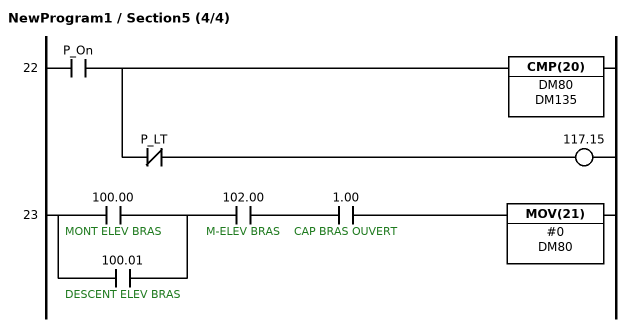
; [picture p24: NewProgram1 / Section5, rungs 22-23]
; rung 22
LD P_On
CMP(20) DM80 DM135
ANDNOT P_LT
OUT 117.15
; rung 23
LD 100.00  ; MONT ELEV BRAS
OR 100.01  ; DESCENT ELEV BRAS
AND 102.00  ; M-ELEV BRAS
AND 1.00  ; CAP BRAS OUVERT
MOV(21) #0 DM80

### Section Section6

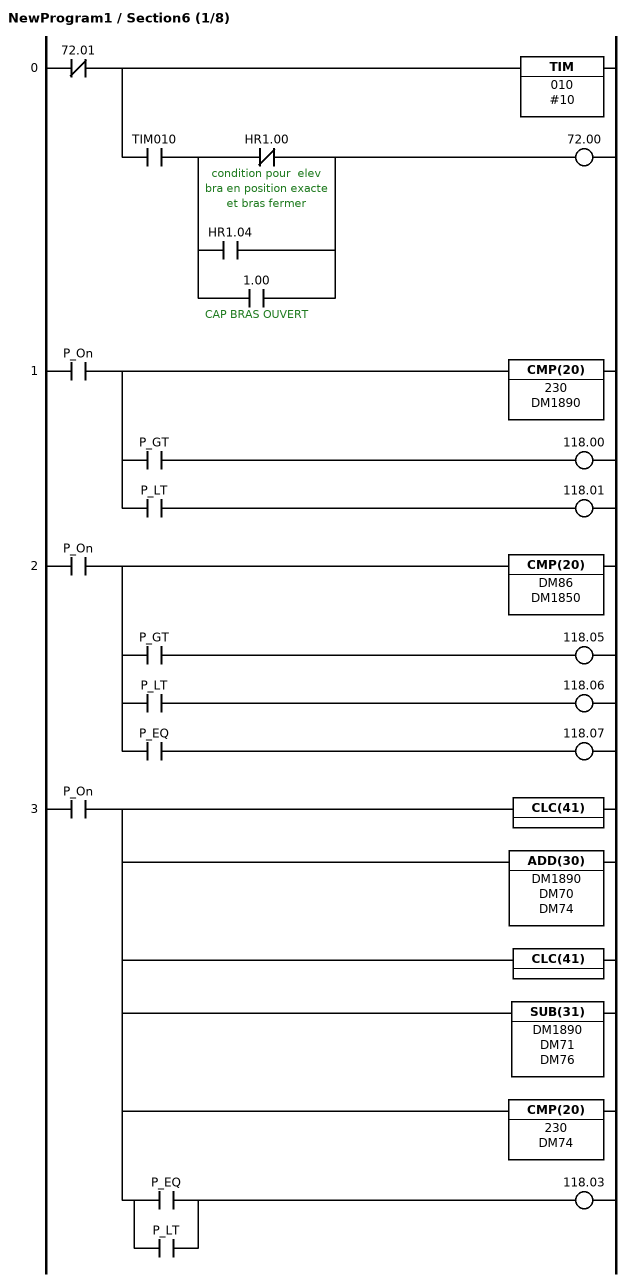
; rung 0
LDNOT 72.01
TIM 010 #10
AND TIM010
LDNOT HR1.00  ; condition pour  elev bra en position exacte et bras fermer
OR HR1.04
OR 1.00  ; CAP BRAS OUVERT
ANDLD
OUT 72.00
; rung 1
LD P_On
OUT TR0
CMP(20) 230 DM1890
AND P_GT
OUT 118.00
LD TR0
AND P_LT
OUT 118.01
; rung 2
LD P_On
OUT TR0
CMP(20) DM86 DM1850
AND P_GT
OUT 118.05
LD TR0
AND P_LT
OUT 118.06
LD TR0
AND P_EQ
OUT 118.07
; rung 3
LD P_On
CLC(41)
ADD(30) DM1890 DM70 DM74
CLC(41)
SUB(31) DM1890 DM71 DM76
CMP(20) 230 DM74
LD P_EQ
OR P_LT
ANDLD
OUT 118.03

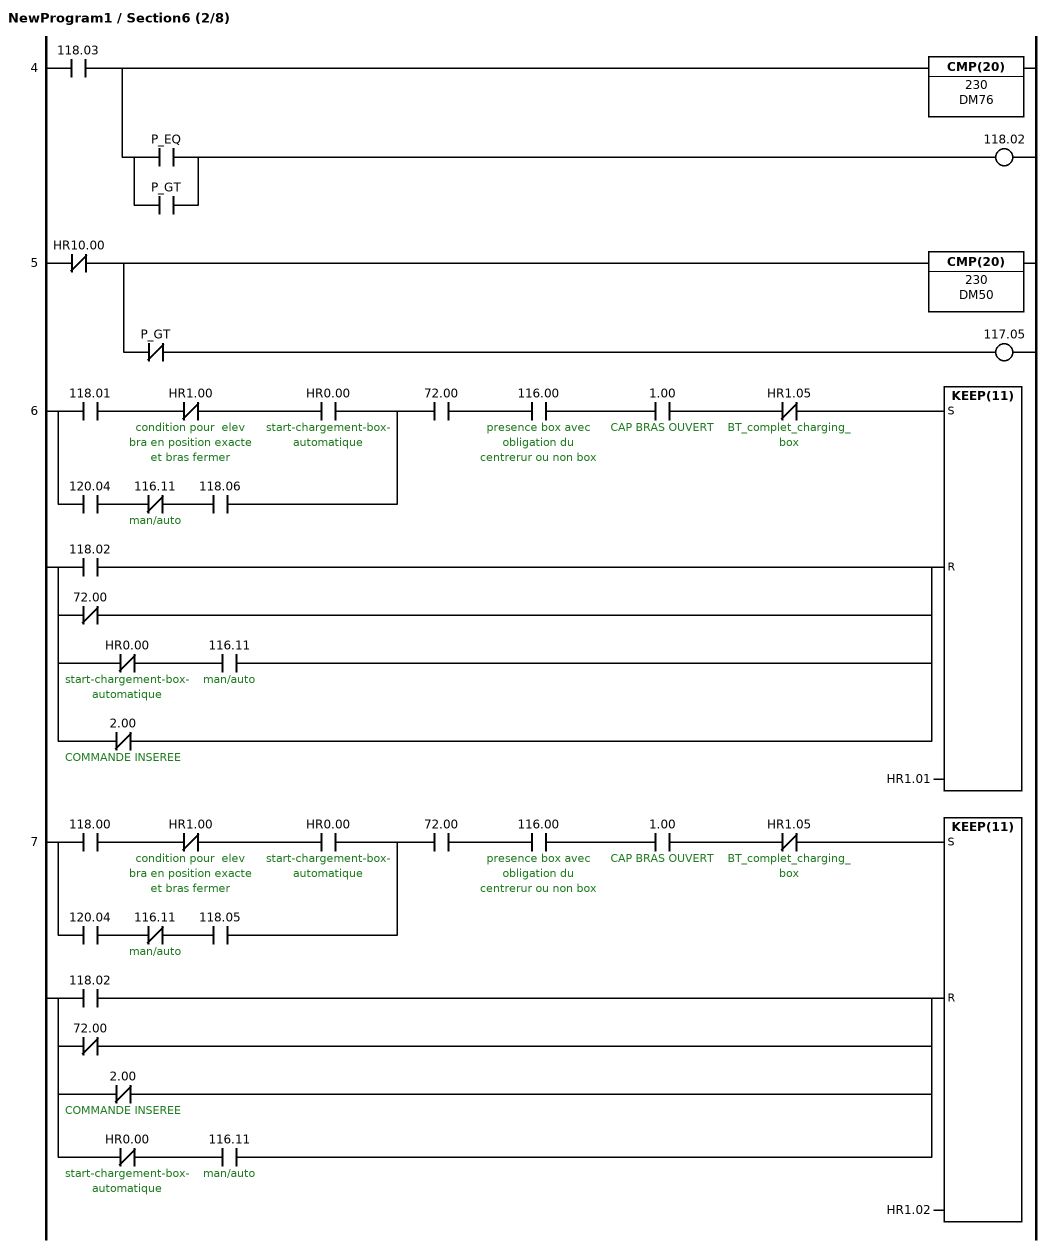
; rung 4
LD 118.03
CMP(20) 230 DM76
LD P_EQ
OR P_GT
ANDLD
OUT 118.02
; rung 5
LDNOT HR10.00
CMP(20) 230 DM50
ANDNOT P_GT
OUT 117.05
; rung 6
LD 118.01
ANDNOT HR1.00  ; condition pour  elev bra en position exacte et bras fermer
AND HR0.00  ; start-chargement-box-automatique
LD 120.04
ANDNOT 116.11  ; man/auto
AND 118.06
ORLD
AND 72.00
AND 116.00  ; presence box avec obligation du centrerur ou non box
AND 1.00  ; CAP BRAS OUVERT
ANDNOT HR1.05  ; BT_complet_charging_box
LD 118.02
ORNOT 72.00
LDNOT HR0.00  ; start-chargement-box-automatique
AND 116.11  ; man/auto
ORLD
ORNOT 2.00  ; COMMANDE INSEREE
KEEP(11) HR1.01
; rung 7
LD 118.00
ANDNOT HR1.00  ; condition pour  elev bra en position exacte et bras fermer
AND HR0.00  ; start-chargement-box-automatique
LD 120.04
ANDNOT 116.11  ; man/auto
AND 118.05
ORLD
AND 72.00
AND 116.00  ; presence box avec obligation du centrerur ou non box
AND 1.00  ; CAP BRAS OUVERT
ANDNOT HR1.05  ; BT_complet_charging_box
LD 118.02
ORNOT 72.00
ORNOT 2.00  ; COMMANDE INSEREE
LDNOT HR0.00  ; start-chargement-box-automatique
AND 116.11  ; man/auto
ORLD
KEEP(11) HR1.02

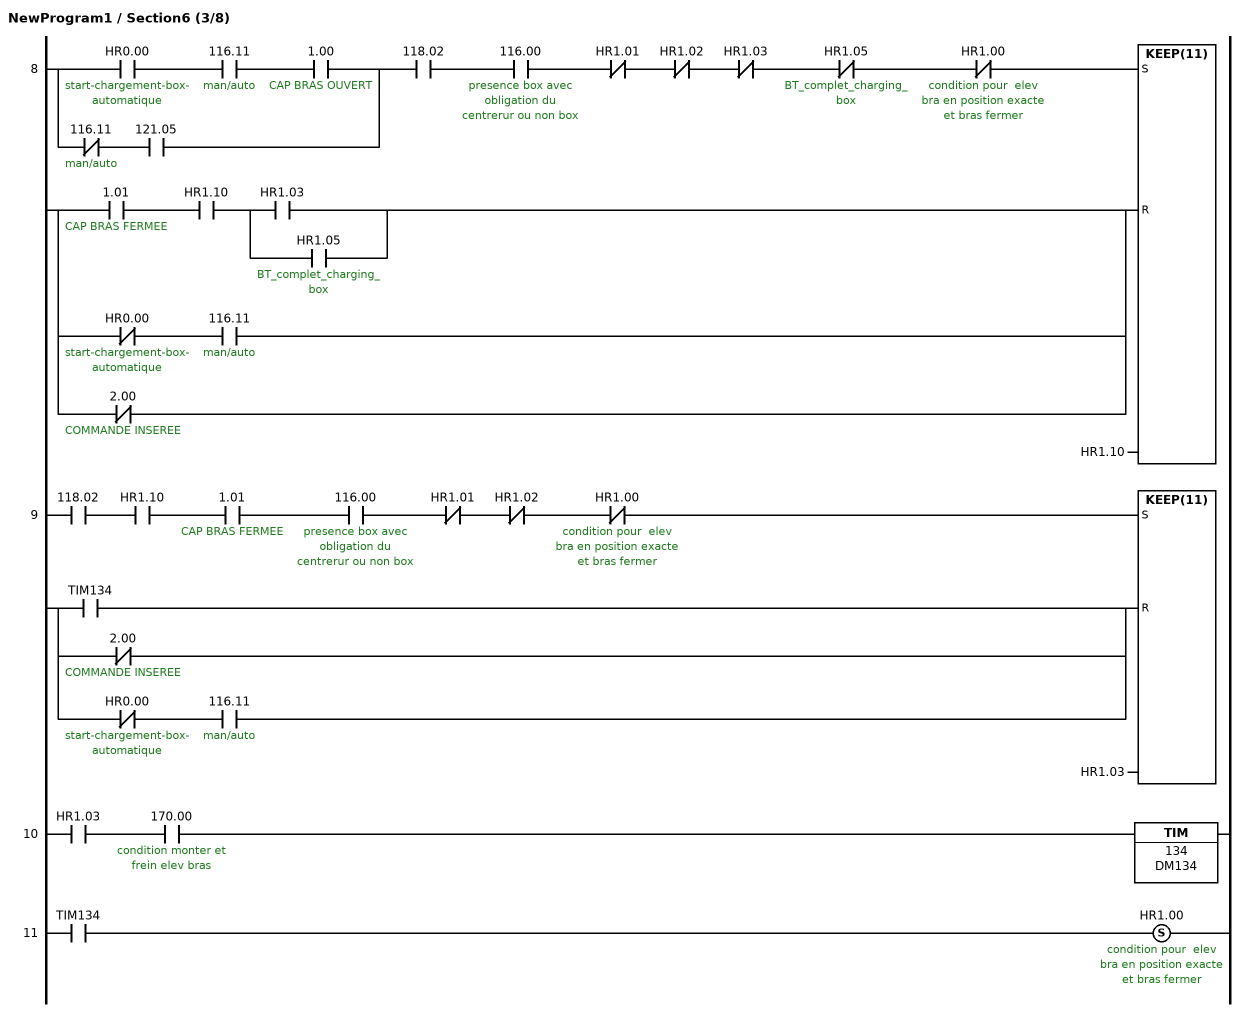
; rung 8
LD HR0.00  ; start-chargement-box-automatique
AND 116.11  ; man/auto
AND 1.00  ; CAP BRAS OUVERT
LDNOT 116.11  ; man/auto
AND 121.05
ORLD
AND 118.02
AND 116.00  ; presence box avec obligation du centrerur ou non box
ANDNOT HR1.01
ANDNOT HR1.02
ANDNOT HR1.03
ANDNOT HR1.05  ; BT_complet_charging_box
ANDNOT HR1.00  ; condition pour  elev bra en position exacte et bras fermer
LD 1.01  ; CAP BRAS FERMEE
AND HR1.10
LD HR1.03
OR HR1.05  ; BT_complet_charging_box
ANDLD
LDNOT HR0.00  ; start-chargement-box-automatique
AND 116.11  ; man/auto
ORLD
ORNOT 2.00  ; COMMANDE INSEREE
KEEP(11) HR1.10
; rung 9
LD 118.02
AND HR1.10
AND 1.01  ; CAP BRAS FERMEE
AND 116.00  ; presence box avec obligation du centrerur ou non box
ANDNOT HR1.01
ANDNOT HR1.02
ANDNOT HR1.00  ; condition pour  elev bra en position exacte et bras fermer
LD TIM134
ORNOT 2.00  ; COMMANDE INSEREE
LDNOT HR0.00  ; start-chargement-box-automatique
AND 116.11  ; man/auto
ORLD
KEEP(11) HR1.03
; rung 10
LD HR1.03
AND 170.00  ; condition monter et frein elev bras
TIM 134 DM134
; rung 11
LD TIM134
SET HR1.00  ; condition pour  elev bra en position exacte et bras fermer

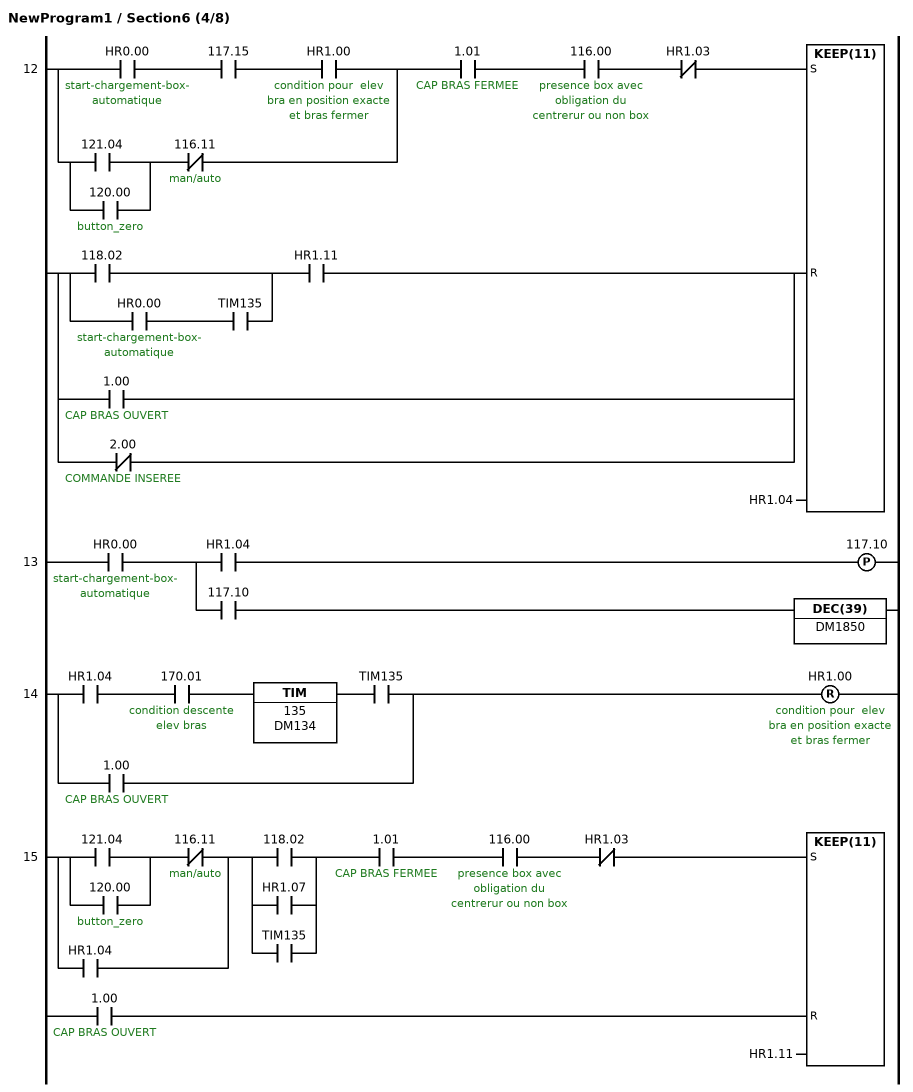
; rung 12
LD HR0.00  ; start-chargement-box-automatique
AND 117.15
AND HR1.00  ; condition pour  elev bra en position exacte et bras fermer
LD 121.04
OR 120.00  ; button_zero
ANDNOT 116.11  ; man/auto
ORLD
AND 1.01  ; CAP BRAS FERMEE
AND 116.00  ; presence box avec obligation du centrerur ou non box
ANDNOT HR1.03
LD 118.02
LD HR0.00  ; start-chargement-box-automatique
AND TIM135
ORLD
AND HR1.11
OR 1.00  ; CAP BRAS OUVERT
ORNOT 2.00  ; COMMANDE INSEREE
KEEP(11) HR1.04
; rung 13
LD HR0.00  ; start-chargement-box-automatique
OUT TR0
AND HR1.04
DIFU(13) 117.10
LD TR0
AND 117.10
DEC(39) DM1850
; rung 14
LD HR1.04
AND 170.01  ; condition descente elev bras
TIM 135 DM134
AND TIM135
OR 1.00  ; CAP BRAS OUVERT
RSET HR1.00  ; condition pour  elev bra en position exacte et bras fermer
; rung 15
LD 121.04
OR 120.00  ; button_zero
ANDNOT 116.11  ; man/auto
OR HR1.04
LD 118.02
OR HR1.07
OR TIM135
ANDLD
AND 1.01  ; CAP BRAS FERMEE
AND 116.00  ; presence box avec obligation du centrerur ou non box
ANDNOT HR1.03
LD 1.00  ; CAP BRAS OUVERT
KEEP(11) HR1.11

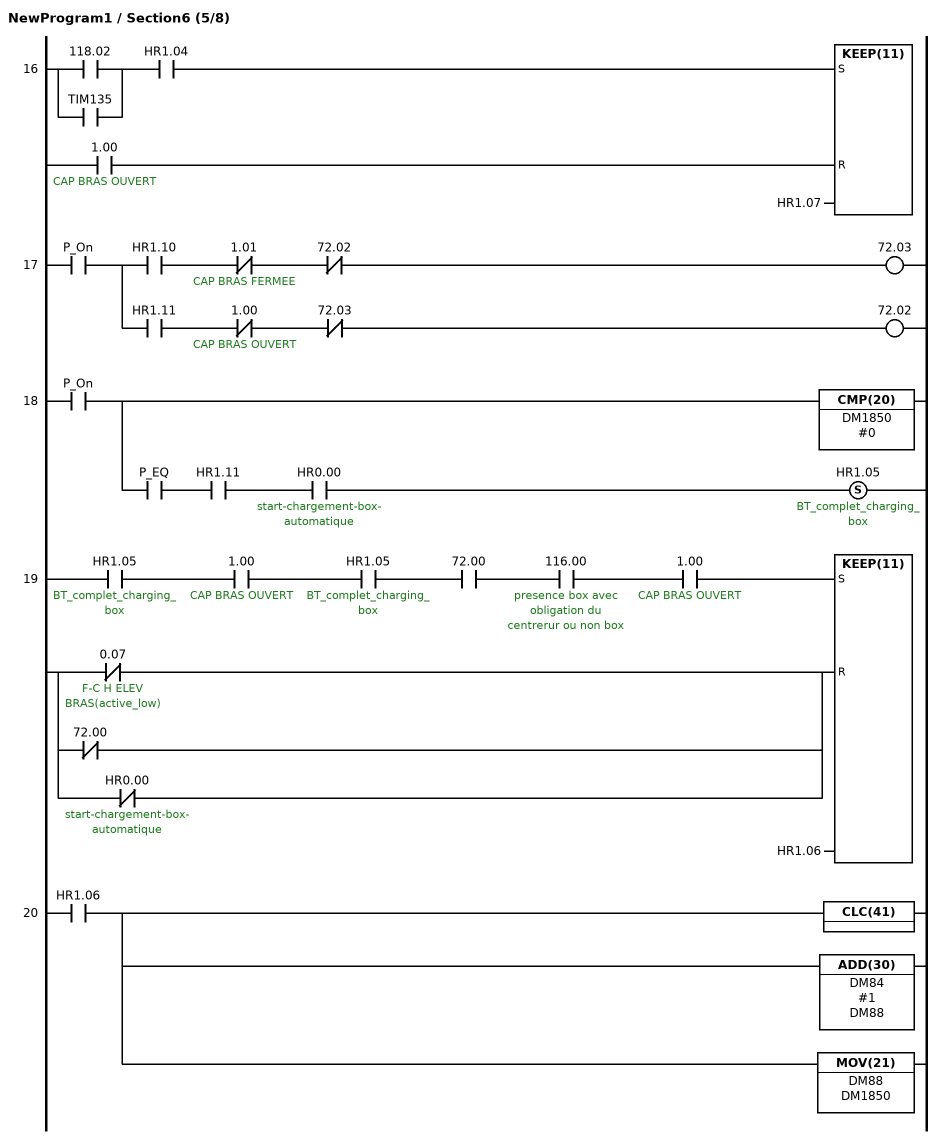
; rung 16
LD 118.02
OR TIM135
AND HR1.04
LD 1.00  ; CAP BRAS OUVERT
KEEP(11) HR1.07
; rung 17
LD P_On
OUT TR0
AND HR1.10
ANDNOT 1.01  ; CAP BRAS FERMEE
ANDNOT 72.02
OUT 72.03
LD TR0
AND HR1.11
ANDNOT 1.00  ; CAP BRAS OUVERT
ANDNOT 72.03
OUT 72.02
; rung 18
LD P_On
CMP(20) DM1850 #0
AND P_EQ
AND HR1.11
AND HR0.00  ; start-chargement-box-automatique
SET HR1.05  ; BT_complet_charging_box
; rung 19
LD HR1.05  ; BT_complet_charging_box
AND 1.00  ; CAP BRAS OUVERT
AND HR1.05  ; BT_complet_charging_box
AND 72.00
AND 116.00  ; presence box avec obligation du centrerur ou non box
AND 1.00  ; CAP BRAS OUVERT
LDNOT 0.07  ; F-C H ELEV BRAS(active_low)
ORNOT 72.00
ORNOT HR0.00  ; start-chargement-box-automatique
KEEP(11) HR1.06
; rung 20
LD HR1.06
CLC(41)
ADD(30) DM84 #1 DM88
MOV(21) DM88 DM1850

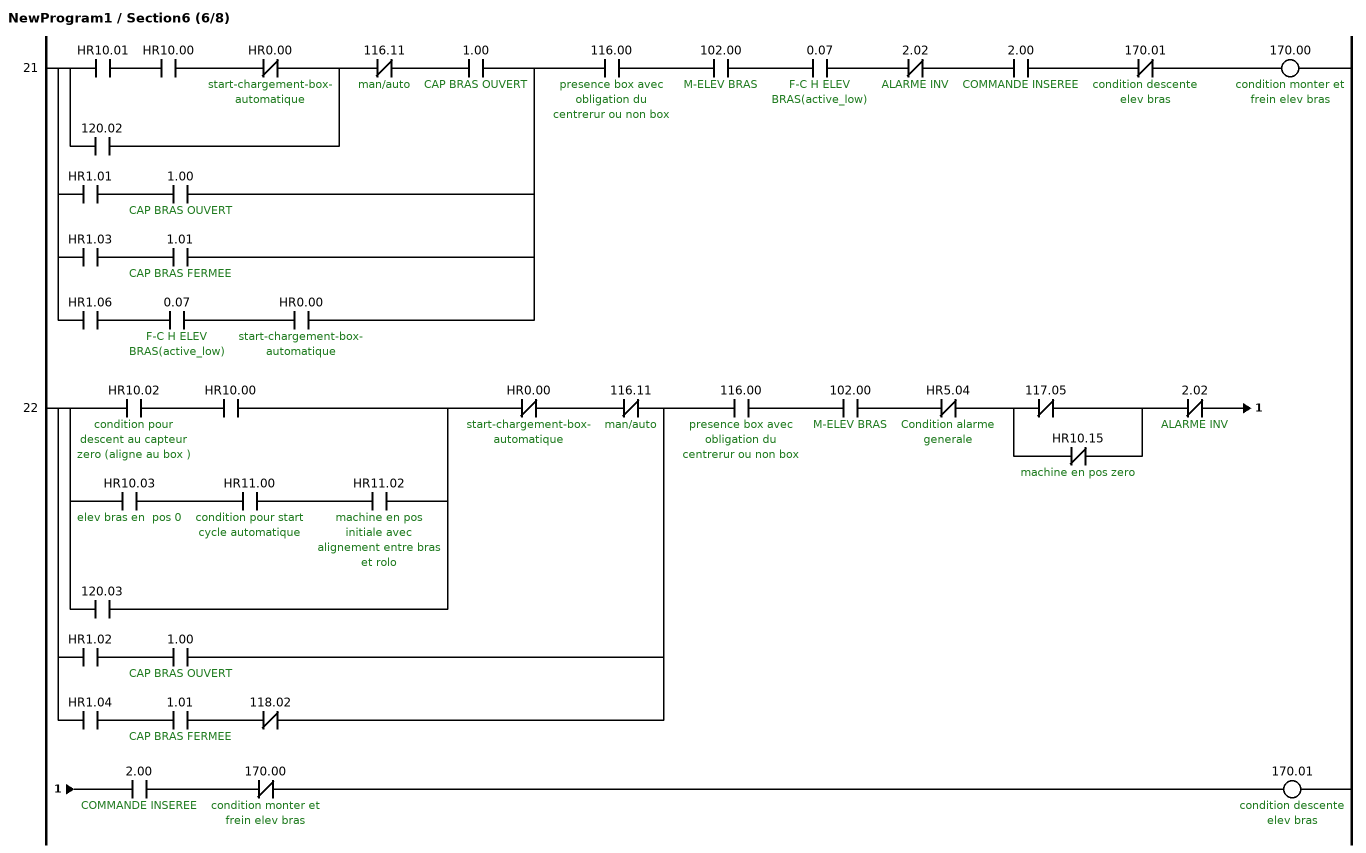
; rung 21
LD HR10.01
AND HR10.00
ANDNOT HR0.00  ; start-chargement-box-automatique
OR 120.02
ANDNOT 116.11  ; man/auto
AND 1.00  ; CAP BRAS OUVERT
LD HR1.01
AND 1.00  ; CAP BRAS OUVERT
ORLD
LD HR1.03
AND 1.01  ; CAP BRAS FERMEE
ORLD
LD HR1.06
AND 0.07  ; F-C H ELEV BRAS(active_low)
AND HR0.00  ; start-chargement-box-automatique
ORLD
AND 116.00  ; presence box avec obligation du centrerur ou non box
AND 102.00  ; M-ELEV BRAS
AND 0.07  ; F-C H ELEV BRAS(active_low)
ANDNOT 2.02  ; ALARME INV
AND 2.00  ; COMMANDE INSEREE
ANDNOT 170.01  ; condition descente elev bras
OUT 170.00  ; condition monter et frein elev bras
; rung 22
LD HR10.02  ; condition pour descent au capteur zero (aligne au box )
AND HR10.00
LD HR10.03  ; elev bras en  pos 0
AND HR11.00  ; condition pour start cycle automatique
AND HR11.02  ; machine en pos initiale avec alignement entre bras et rolo
ORLD
OR 120.03
ANDNOT HR0.00  ; start-chargement-box-automatique
ANDNOT 116.11  ; man/auto
LD HR1.02
AND 1.00  ; CAP BRAS OUVERT
ORLD
LD HR1.04
AND 1.01  ; CAP BRAS FERMEE
ANDNOT 118.02
ORLD
AND 116.00  ; presence box avec obligation du centrerur ou non box
AND 102.00  ; M-ELEV BRAS
ANDNOT HR5.04  ; Condition alarme generale
LDNOT 117.05
ORNOT HR10.15  ; machine en pos zero
ANDLD
ANDNOT 2.02  ; ALARME INV
AND 2.00  ; COMMANDE INSEREE
ANDNOT 170.00  ; condition monter et frein elev bras
OUT 170.01  ; condition descente elev bras

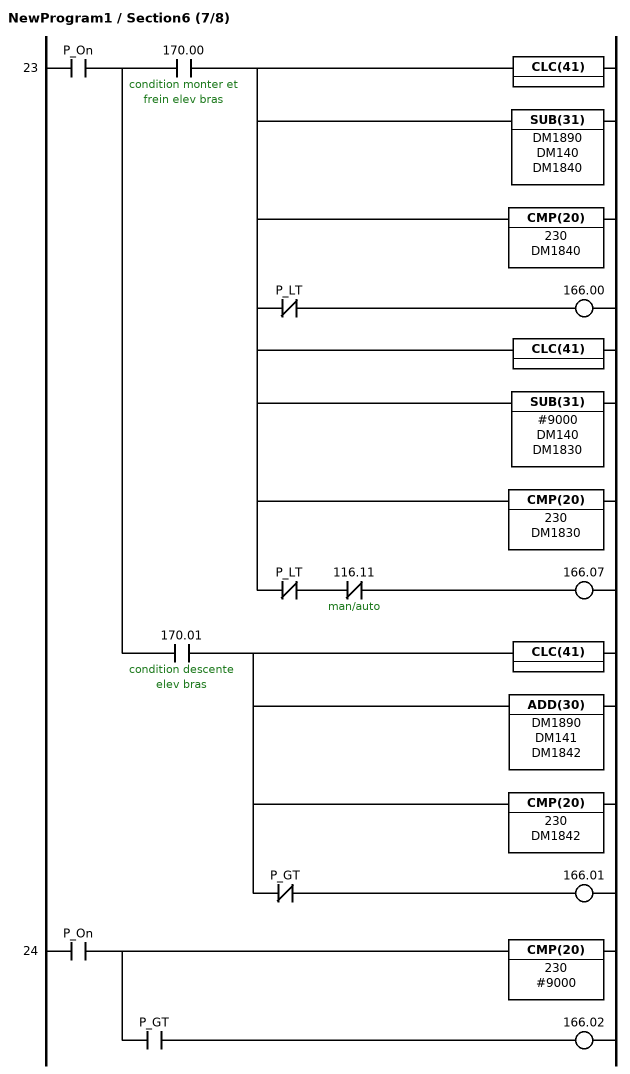
; rung 23
LD P_On
OUT TR0
AND 170.00  ; condition monter et frein elev bras
OUT TR1
CLC(41)
SUB(31) DM1890 DM140 DM1840
CMP(20) 230 DM1840
ANDNOT P_LT
OUT 166.00
LD TR1
CLC(41)
SUB(31) #9000 DM140 DM1830
CMP(20) 230 DM1830
ANDNOT P_LT
ANDNOT 116.11  ; man/auto
OUT 166.07
LD TR0
AND 170.01  ; condition descente elev bras
CLC(41)
ADD(30) DM1890 DM141 DM1842
CMP(20) 230 DM1842
ANDNOT P_GT
OUT 166.01
; rung 24
LD P_On
CMP(20) 230 #9000
AND P_GT
OUT 166.02

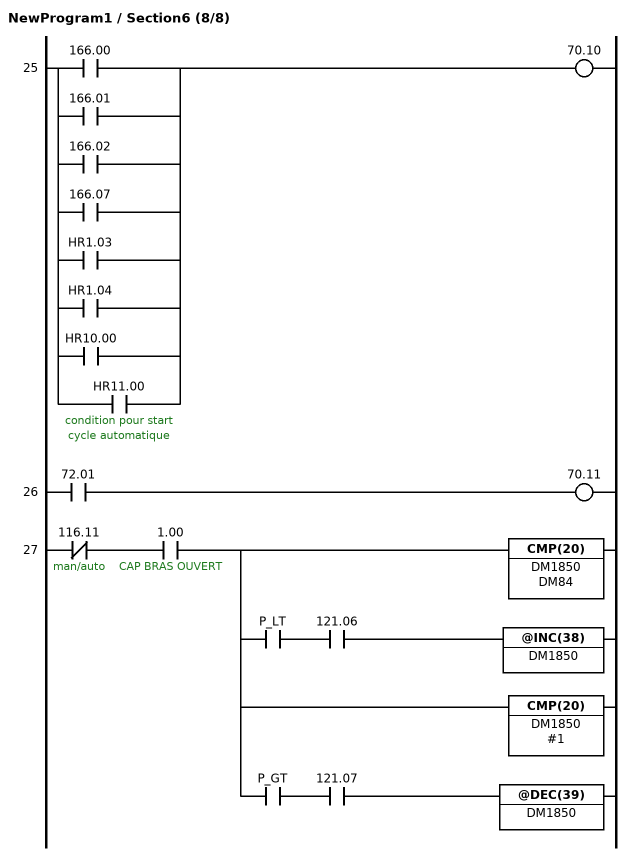
; rung 25
LD 166.00
OR 166.01
OR 166.02
OR 166.07
OR HR1.03
OR HR1.04
OR HR10.00
OR HR11.00  ; condition pour start cycle automatique
OUT 70.10
; rung 26
LD 72.01
OUT 70.11
; rung 27
LDNOT 116.11  ; man/auto
AND 1.00  ; CAP BRAS OUVERT
OUT TR0
CMP(20) DM1850 DM84
AND P_LT
AND 121.06
@INC(38) DM1850
LD TR0
CMP(20) DM1850 #1
AND P_GT
AND 121.07
@DEC(39) DM1850

### Section Section7

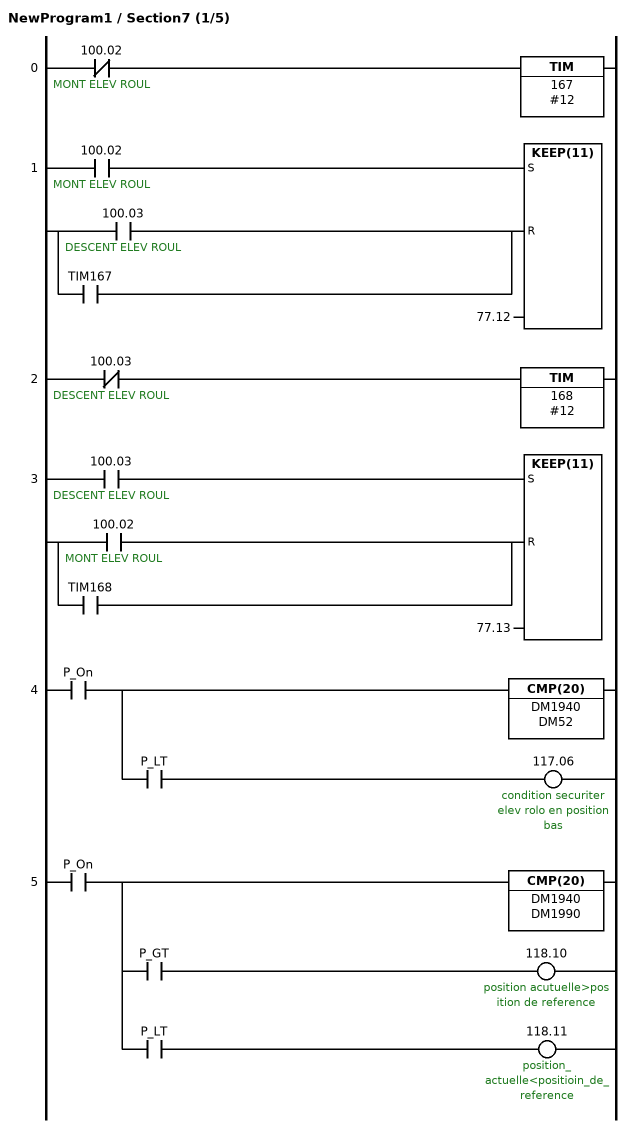
; rung 0
LDNOT 100.02  ; MONT ELEV ROUL
TIM 167 #12
; rung 1
LD 100.02  ; MONT ELEV ROUL
LD 100.03  ; DESCENT ELEV ROUL
OR TIM167
KEEP(11) 77.12
; rung 2
LDNOT 100.03  ; DESCENT ELEV ROUL
TIM 168 #12
; rung 3
LD 100.03  ; DESCENT ELEV ROUL
LD 100.02  ; MONT ELEV ROUL
OR TIM168
KEEP(11) 77.13
; rung 4
LD P_On
CMP(20) DM1940 DM52
AND P_LT
OUT 117.06  ; condition securiter elev rolo en position bas
; rung 5
LD P_On
OUT TR0
CMP(20) DM1940 DM1990
AND P_GT
OUT 118.10  ; position acutuelle>position de reference
LD TR0
AND P_LT
OUT 118.11  ; position_actuelle<positioin_de_reference

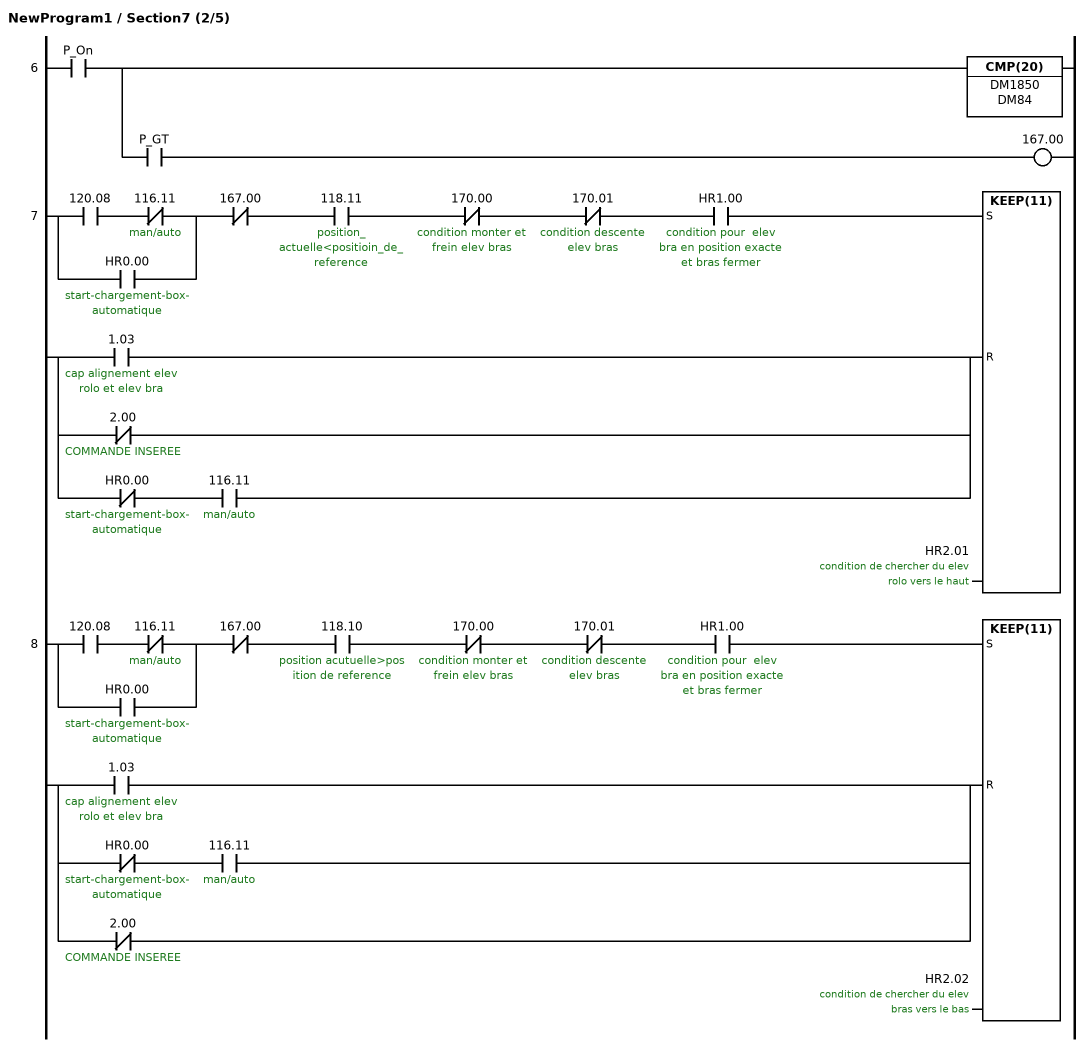
; rung 6
LD P_On
CMP(20) DM1850 DM84
AND P_GT
OUT 167.00
; rung 7
LD 120.08
ANDNOT 116.11  ; man/auto
OR HR0.00  ; start-chargement-box-automatique
ANDNOT 167.00
AND 118.11  ; position_actuelle<positioin_de_reference
ANDNOT 170.00  ; condition monter et frein elev bras
ANDNOT 170.01  ; condition descente elev bras
AND HR1.00  ; condition pour  elev bra en position exacte et bras fermer
LD 1.03  ; cap alignement elev rolo et elev bra
ORNOT 2.00  ; COMMANDE INSEREE
LDNOT HR0.00  ; start-chargement-box-automatique
AND 116.11  ; man/auto
ORLD
KEEP(11) HR2.01  ; condition de chercher du elev rolo vers le haut
; rung 8
LD 120.08
ANDNOT 116.11  ; man/auto
OR HR0.00  ; start-chargement-box-automatique
ANDNOT 167.00
AND 118.10  ; position acutuelle>position de reference
ANDNOT 170.00  ; condition monter et frein elev bras
ANDNOT 170.01  ; condition descente elev bras
AND HR1.00  ; condition pour  elev bra en position exacte et bras fermer
LD 1.03  ; cap alignement elev rolo et elev bra
LDNOT HR0.00  ; start-chargement-box-automatique
AND 116.11  ; man/auto
ORLD
ORNOT 2.00  ; COMMANDE INSEREE
KEEP(11) HR2.02  ; condition de chercher du elev bras vers le bas

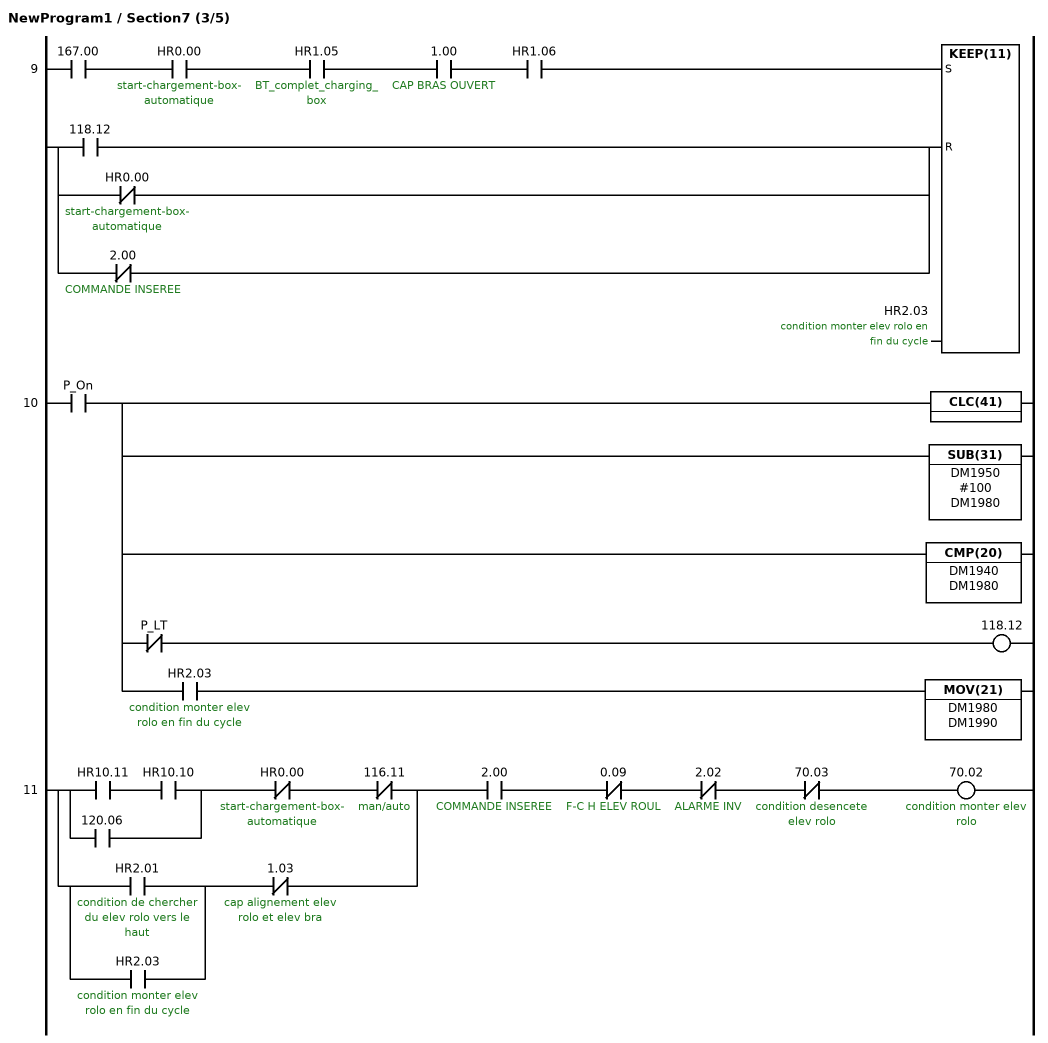
; rung 9
LD 167.00
AND HR0.00  ; start-chargement-box-automatique
AND HR1.05  ; BT_complet_charging_box
AND 1.00  ; CAP BRAS OUVERT
AND HR1.06
LD 118.12
ORNOT HR0.00  ; start-chargement-box-automatique
ORNOT 2.00  ; COMMANDE INSEREE
KEEP(11) HR2.03  ; condition monter elev rolo en fin du cycle
; rung 10
LD P_On
OUT TR0
CLC(41)
SUB(31) DM1950 #100 DM1980
CMP(20) DM1940 DM1980
ANDNOT P_LT
OUT 118.12
LD TR0
AND HR2.03  ; condition monter elev rolo en fin du cycle
MOV(21) DM1980 DM1990
; rung 11
LD HR10.11
AND HR10.10
OR 120.06
ANDNOT HR0.00  ; start-chargement-box-automatique
ANDNOT 116.11  ; man/auto
LD HR2.01  ; condition de chercher du elev rolo vers le haut
OR HR2.03  ; condition monter elev rolo en fin du cycle
ANDNOT 1.03  ; cap alignement elev rolo et elev bra
ORLD
AND 2.00  ; COMMANDE INSEREE
ANDNOT 0.09  ; F-C H ELEV ROUL
ANDNOT 2.02  ; ALARME INV
ANDNOT 70.03  ; condition desencete elev rolo
OUT 70.02  ; condition monter elev rolo

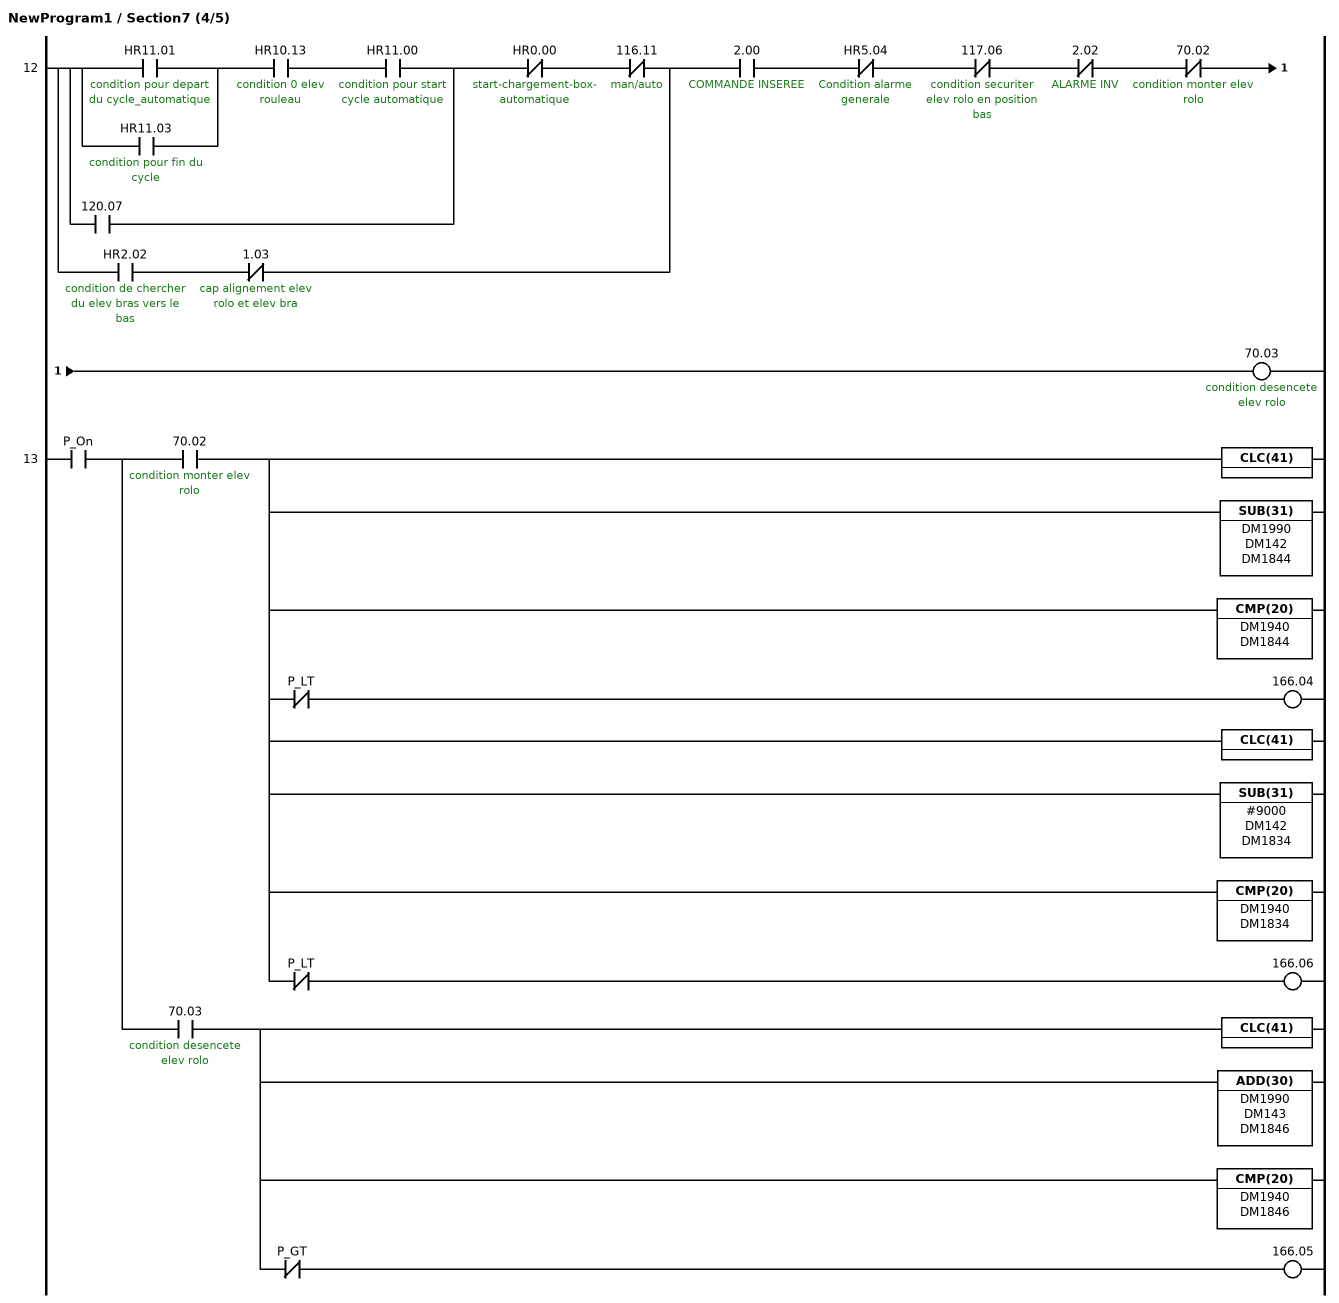
; rung 12
LD HR11.01  ; condition pour depart du cycle_automatique
OR HR11.03  ; condition pour fin du cycle
AND HR10.13  ; condition 0 elev rouleau
AND HR11.00  ; condition pour start cycle automatique
OR 120.07
ANDNOT HR0.00  ; start-chargement-box-automatique
ANDNOT 116.11  ; man/auto
LD HR2.02  ; condition de chercher du elev bras vers le bas
ANDNOT 1.03  ; cap alignement elev rolo et elev bra
ORLD
AND 2.00  ; COMMANDE INSEREE
ANDNOT HR5.04  ; Condition alarme generale
ANDNOT 117.06  ; condition securiter elev rolo en position bas
ANDNOT 2.02  ; ALARME INV
ANDNOT 70.02  ; condition monter elev rolo
OUT 70.03  ; condition desencete elev rolo
; rung 13
LD P_On
OUT TR0
AND 70.02  ; condition monter elev rolo
OUT TR1
CLC(41)
SUB(31) DM1990 DM142 DM1844
CMP(20) DM1940 DM1844
ANDNOT P_LT
OUT 166.04
LD TR1
CLC(41)
SUB(31) #9000 DM142 DM1834
CMP(20) DM1940 DM1834
ANDNOT P_LT
OUT 166.06
LD TR0
AND 70.03  ; condition desencete elev rolo
CLC(41)
ADD(30) DM1990 DM143 DM1846
CMP(20) DM1940 DM1846
ANDNOT P_GT
OUT 166.05

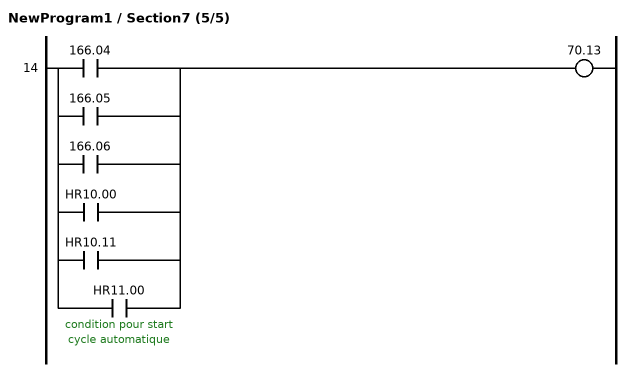
; rung 14
LD 166.04
OR 166.05
OR 166.06
OR HR10.00
OR HR10.11
OR HR11.00  ; condition pour start cycle automatique
OUT 70.13

### Section Section8

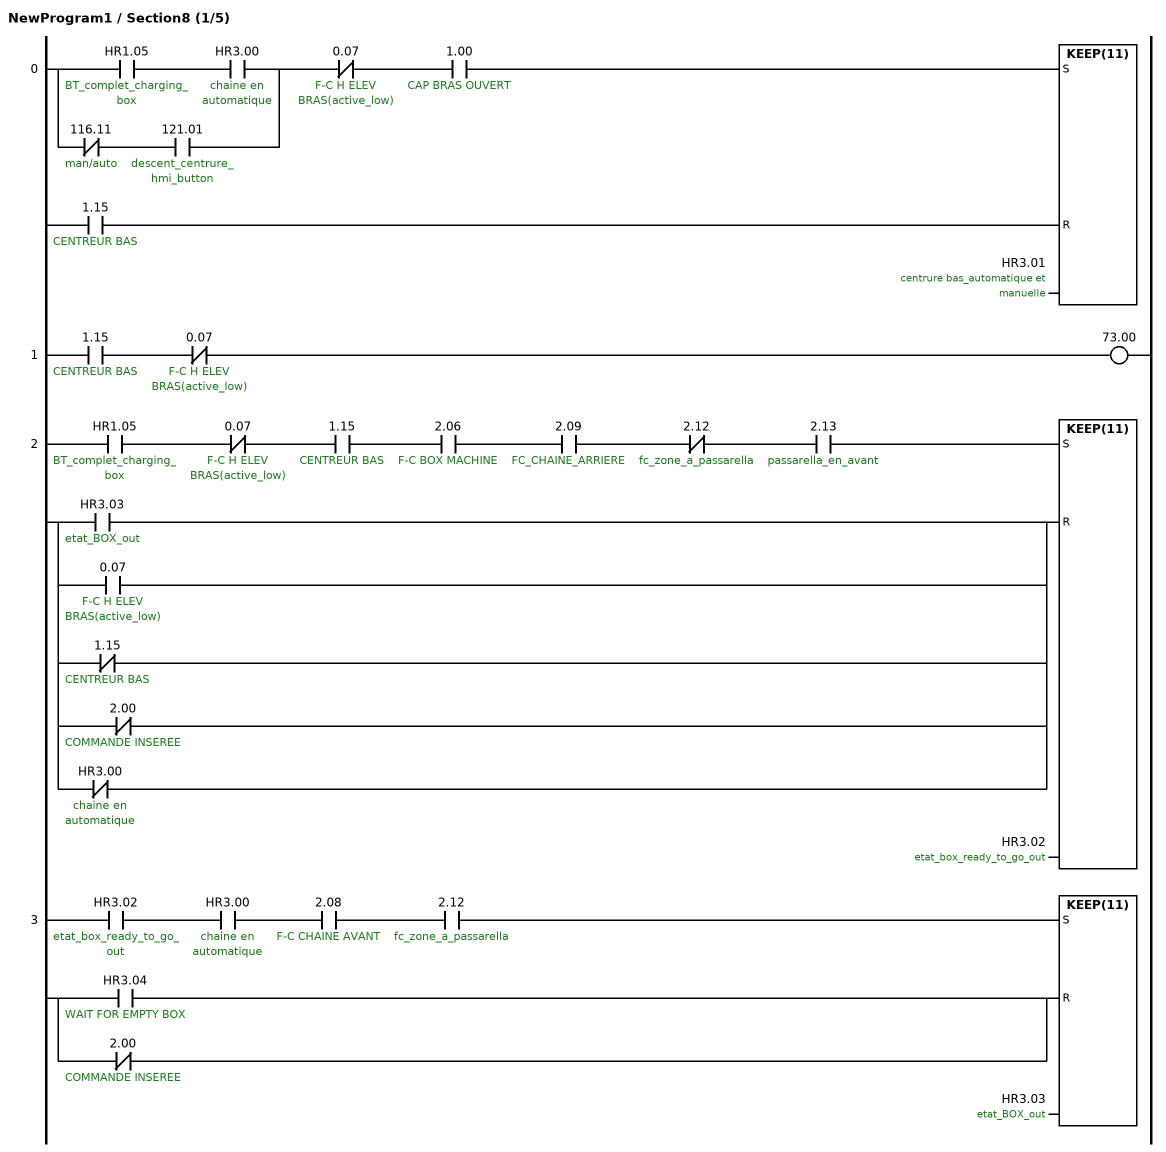
; rung 0
LD HR1.05  ; BT_complet_charging_box
AND HR3.00  ; chaine en automatique
LDNOT 116.11  ; man/auto
AND 121.01  ; descent_centrure_hmi_button
ORLD
ANDNOT 0.07  ; F-C H ELEV BRAS(active_low)
AND 1.00  ; CAP BRAS OUVERT
LD 1.15  ; CENTREUR BAS
KEEP(11) HR3.01  ; centrure bas_automatique et manuelle
; rung 1
LD 1.15  ; CENTREUR BAS
ANDNOT 0.07  ; F-C H ELEV BRAS(active_low)
OUT 73.00
; rung 2
LD HR1.05  ; BT_complet_charging_box
ANDNOT 0.07  ; F-C H ELEV BRAS(active_low)
AND 1.15  ; CENTREUR BAS
AND 2.06  ; F-C BOX MACHINE
AND 2.09  ; FC_CHAINE_ARRIERE
ANDNOT 2.12  ; fc_zone_a_passarella
AND 2.13  ; passarella_en_avant
LD HR3.03  ; etat_BOX_out
OR 0.07  ; F-C H ELEV BRAS(active_low)
ORNOT 1.15  ; CENTREUR BAS
ORNOT 2.00  ; COMMANDE INSEREE
ORNOT HR3.00  ; chaine en automatique
KEEP(11) HR3.02  ; etat_box_ready_to_go_out
; rung 3
LD HR3.02  ; etat_box_ready_to_go_out
AND HR3.00  ; chaine en automatique
AND 2.08  ; F-C CHAINE AVANT
AND 2.12  ; fc_zone_a_passarella
LD HR3.04  ; WAIT FOR EMPTY BOX
ORNOT 2.00  ; COMMANDE INSEREE
KEEP(11) HR3.03  ; etat_BOX_out

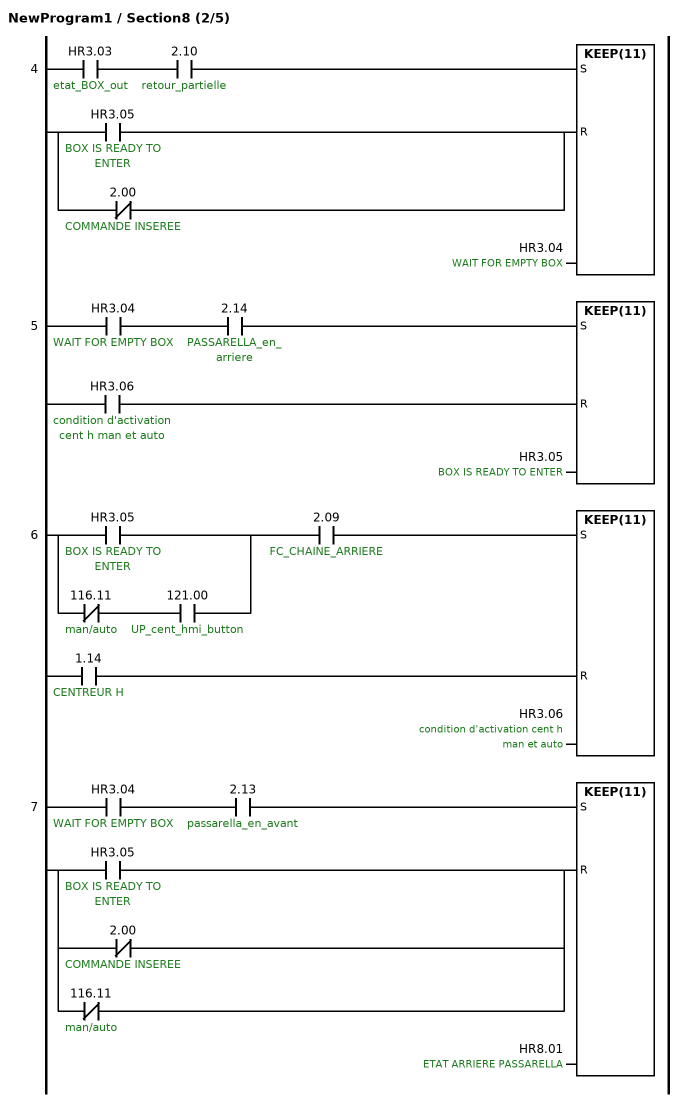
; rung 4
LD HR3.03  ; etat_BOX_out
AND 2.10  ; retour_partielle
LD HR3.05  ; BOX IS READY TO ENTER
ORNOT 2.00  ; COMMANDE INSEREE
KEEP(11) HR3.04  ; WAIT FOR EMPTY BOX
; rung 5
LD HR3.04  ; WAIT FOR EMPTY BOX
AND 2.14  ; PASSARELLA_en_arriere
LD HR3.06  ; condition d'activation cent h man et auto
KEEP(11) HR3.05  ; BOX IS READY TO ENTER
; rung 6
LD HR3.05  ; BOX IS READY TO ENTER
LDNOT 116.11  ; man/auto
AND 121.00  ; UP_cent_hmi_button
ORLD
AND 2.09  ; FC_CHAINE_ARRIERE
LD 1.14  ; CENTREUR H
KEEP(11) HR3.06  ; condition d'activation cent h man et auto
; rung 7
LD HR3.04  ; WAIT FOR EMPTY BOX
AND 2.13  ; passarella_en_avant
LD HR3.05  ; BOX IS READY TO ENTER
ORNOT 2.00  ; COMMANDE INSEREE
ORNOT 116.11  ; man/auto
KEEP(11) HR8.01  ; ETAT ARRIERE PASSARELLA

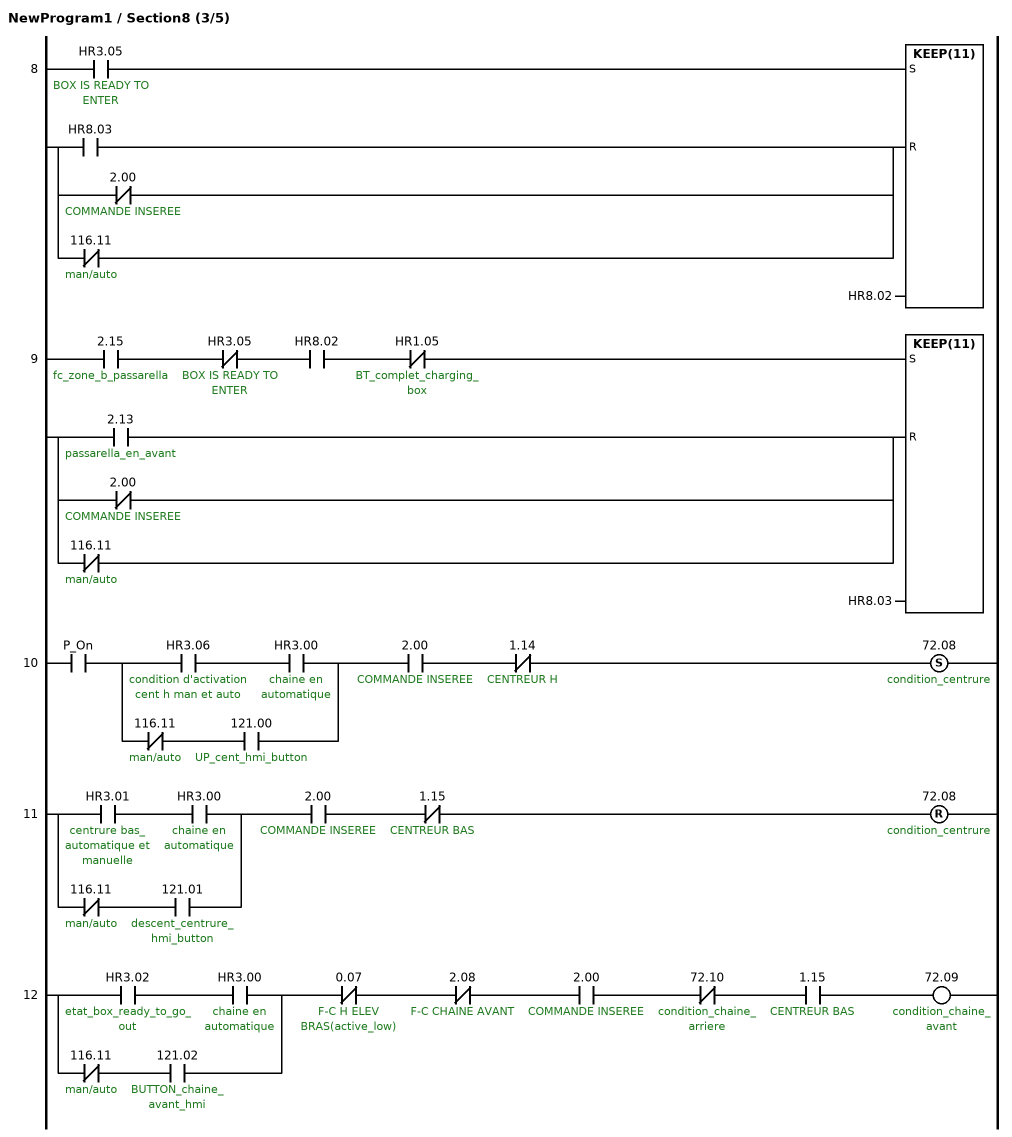
; rung 8
LD HR3.05  ; BOX IS READY TO ENTER
LD HR8.03
ORNOT 2.00  ; COMMANDE INSEREE
ORNOT 116.11  ; man/auto
KEEP(11) HR8.02
; rung 9
LD 2.15  ; fc_zone_b_passarella
ANDNOT HR3.05  ; BOX IS READY TO ENTER
AND HR8.02
ANDNOT HR1.05  ; BT_complet_charging_box
LD 2.13  ; passarella_en_avant
ORNOT 2.00  ; COMMANDE INSEREE
ORNOT 116.11  ; man/auto
KEEP(11) HR8.03
; rung 10
LD P_On
LD HR3.06  ; condition d'activation cent h man et auto
AND HR3.00  ; chaine en automatique
LDNOT 116.11  ; man/auto
AND 121.00  ; UP_cent_hmi_button
ORLD
ANDLD
AND 2.00  ; COMMANDE INSEREE
ANDNOT 1.14  ; CENTREUR H
SET 72.08  ; condition_centrure
; rung 11
LD HR3.01  ; centrure bas_automatique et manuelle
AND HR3.00  ; chaine en automatique
LDNOT 116.11  ; man/auto
AND 121.01  ; descent_centrure_hmi_button
ORLD
AND 2.00  ; COMMANDE INSEREE
ANDNOT 1.15  ; CENTREUR BAS
RSET 72.08  ; condition_centrure
; rung 12
LD HR3.02  ; etat_box_ready_to_go_out
AND HR3.00  ; chaine en automatique
LDNOT 116.11  ; man/auto
AND 121.02  ; BUTTON_chaine_avant_hmi
ORLD
ANDNOT 0.07  ; F-C H ELEV BRAS(active_low)
ANDNOT 2.08  ; F-C CHAINE AVANT
AND 2.00  ; COMMANDE INSEREE
ANDNOT 72.10  ; condition_chaine_arriere
AND 1.15  ; CENTREUR BAS
OUT 72.09  ; condition_chaine_avant

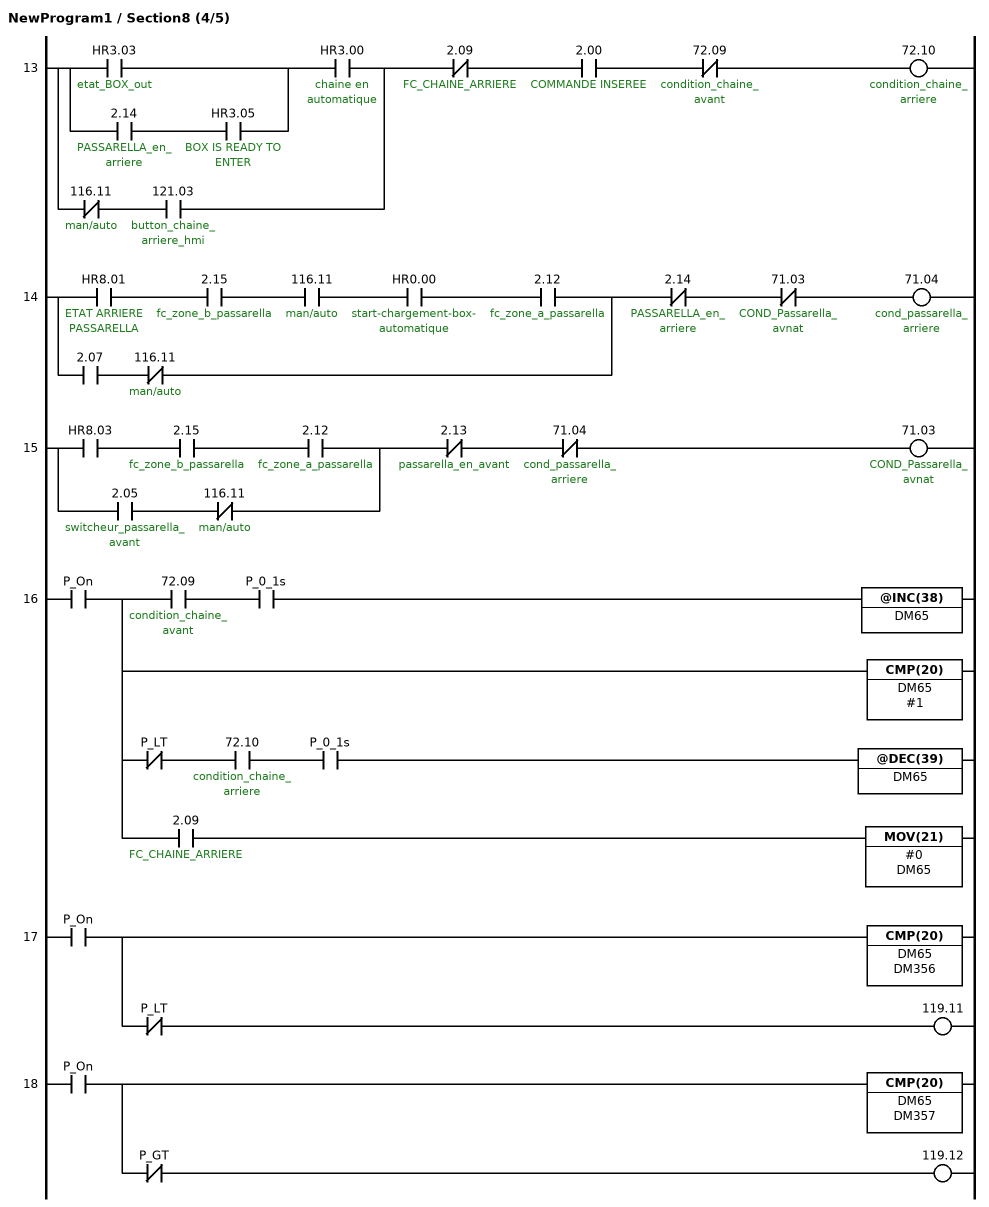
; rung 13
LD HR3.03  ; etat_BOX_out
LD 2.14  ; PASSARELLA_en_arriere
AND HR3.05  ; BOX IS READY TO ENTER
ORLD
AND HR3.00  ; chaine en automatique
LDNOT 116.11  ; man/auto
AND 121.03  ; button_chaine_arriere_hmi
ORLD
ANDNOT 2.09  ; FC_CHAINE_ARRIERE
AND 2.00  ; COMMANDE INSEREE
ANDNOT 72.09  ; condition_chaine_avant
OUT 72.10  ; condition_chaine_arriere
; rung 14
LD HR8.01  ; ETAT ARRIERE PASSARELLA
AND 2.15  ; fc_zone_b_passarella
AND 116.11  ; man/auto
AND HR0.00  ; start-chargement-box-automatique
AND 2.12  ; fc_zone_a_passarella
LD 2.07
ANDNOT 116.11  ; man/auto
ORLD
ANDNOT 2.14  ; PASSARELLA_en_arriere
ANDNOT 71.03  ; COND_Passarella_avnat
OUT 71.04  ; cond_passarella_arriere
; rung 15
LD HR8.03
AND 2.15  ; fc_zone_b_passarella
AND 2.12  ; fc_zone_a_passarella
LD 2.05  ; switcheur_passarella_avant
ANDNOT 116.11  ; man/auto
ORLD
ANDNOT 2.13  ; passarella_en_avant
ANDNOT 71.04  ; cond_passarella_arriere
OUT 71.03  ; COND_Passarella_avnat
; rung 16
LD P_On
OUT TR0
AND 72.09  ; condition_chaine_avant
AND P_0_1s
@INC(38) DM65
LD TR0
CMP(20) DM65 #1
ANDNOT P_LT
AND 72.10  ; condition_chaine_arriere
AND P_0_1s
@DEC(39) DM65
LD TR0
AND 2.09  ; FC_CHAINE_ARRIERE
MOV(21) #0 DM65
; rung 17
LD P_On
CMP(20) DM65 DM356
ANDNOT P_LT
OUT 119.11
; rung 18
LD P_On
CMP(20) DM65 DM357
ANDNOT P_GT
OUT 119.12

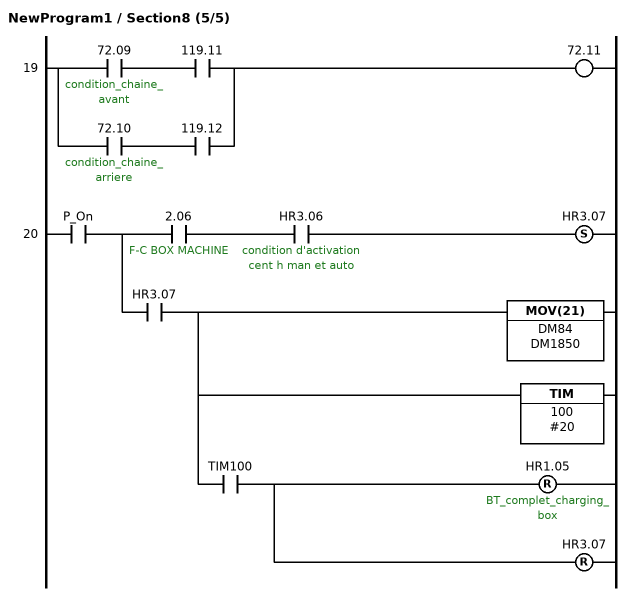
; rung 19
LD 72.09  ; condition_chaine_avant
AND 119.11
LD 72.10  ; condition_chaine_arriere
AND 119.12
ORLD
OUT 72.11
; rung 20
LD P_On
OUT TR0
AND 2.06  ; F-C BOX MACHINE
AND HR3.06  ; condition d'activation cent h man et auto
SET HR3.07
LD TR0
AND HR3.07
MOV(21) DM84 DM1850
TIM 100 #20
AND TIM100
RSET HR1.05  ; BT_complet_charging_box
RSET HR3.07

### Section Section9

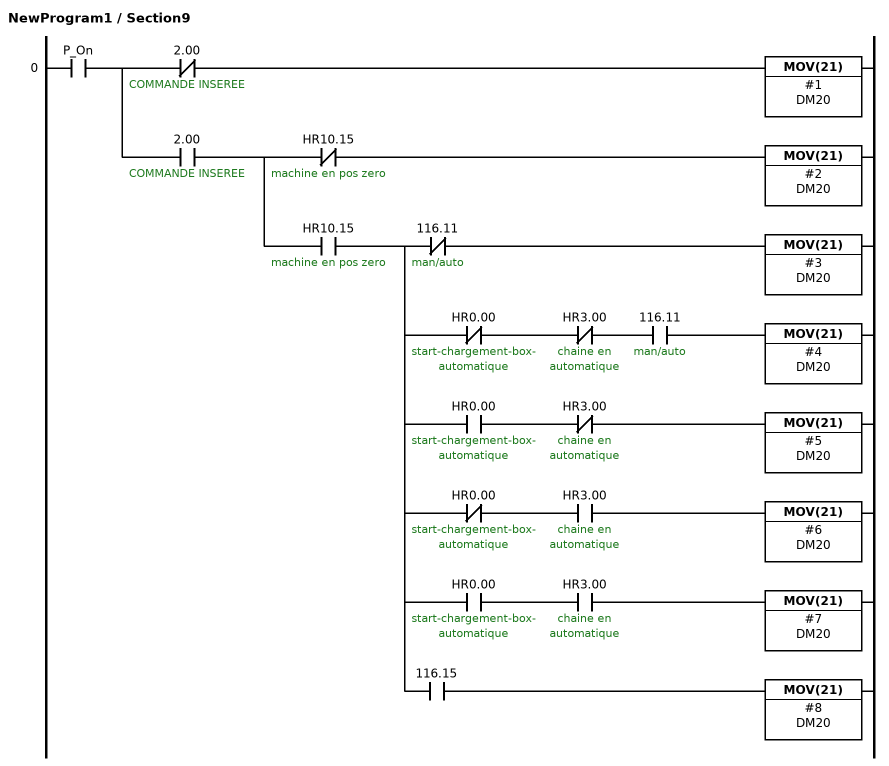
; rung 0
LD P_On
OUT TR0
ANDNOT 2.00  ; COMMANDE INSEREE
MOV(21) #1 DM20
LD TR0
AND 2.00  ; COMMANDE INSEREE
OUT TR0
ANDNOT HR10.15  ; machine en pos zero
MOV(21) #2 DM20
LD TR0
AND HR10.15  ; machine en pos zero
OUT TR0
ANDNOT 116.11  ; man/auto
MOV(21) #3 DM20
LD TR0
ANDNOT HR0.00  ; start-chargement-box-automatique
ANDNOT HR3.00  ; chaine en automatique
AND 116.11  ; man/auto
MOV(21) #4 DM20
LD TR0
AND HR0.00  ; start-chargement-box-automatique
ANDNOT HR3.00  ; chaine en automatique
MOV(21) #5 DM20
LD TR0
ANDNOT HR0.00  ; start-chargement-box-automatique
AND HR3.00  ; chaine en automatique
MOV(21) #6 DM20
LD TR0
AND HR0.00  ; start-chargement-box-automatique
AND HR3.00  ; chaine en automatique
MOV(21) #7 DM20
LD TR0
AND 116.15
MOV(21) #8 DM20

### Section Section10

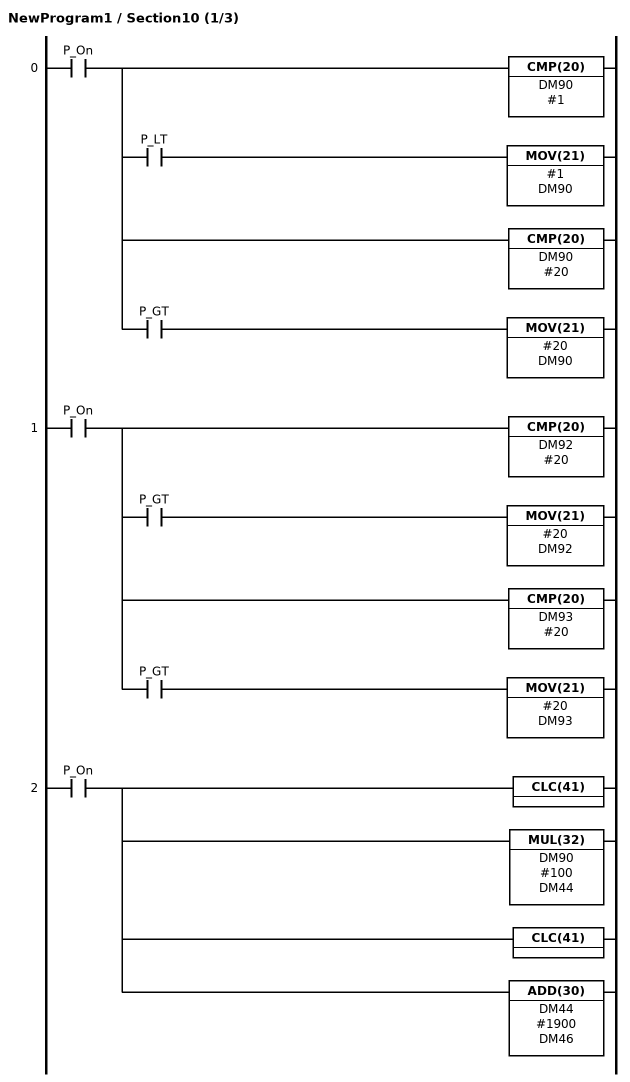
; rung 0
LD P_On
OUT TR0
CMP(20) DM90 #1
AND P_LT
MOV(21) #1 DM90
LD TR0
CMP(20) DM90 #20
AND P_GT
MOV(21) #20 DM90
; rung 1
LD P_On
OUT TR0
CMP(20) DM92 #20
AND P_GT
MOV(21) #20 DM92
LD TR0
CMP(20) DM93 #20
AND P_GT
MOV(21) #20 DM93
; rung 2
LD P_On
CLC(41)
MUL(32) DM90 #100 DM44
CLC(41)
ADD(30) DM44 #1900 DM46

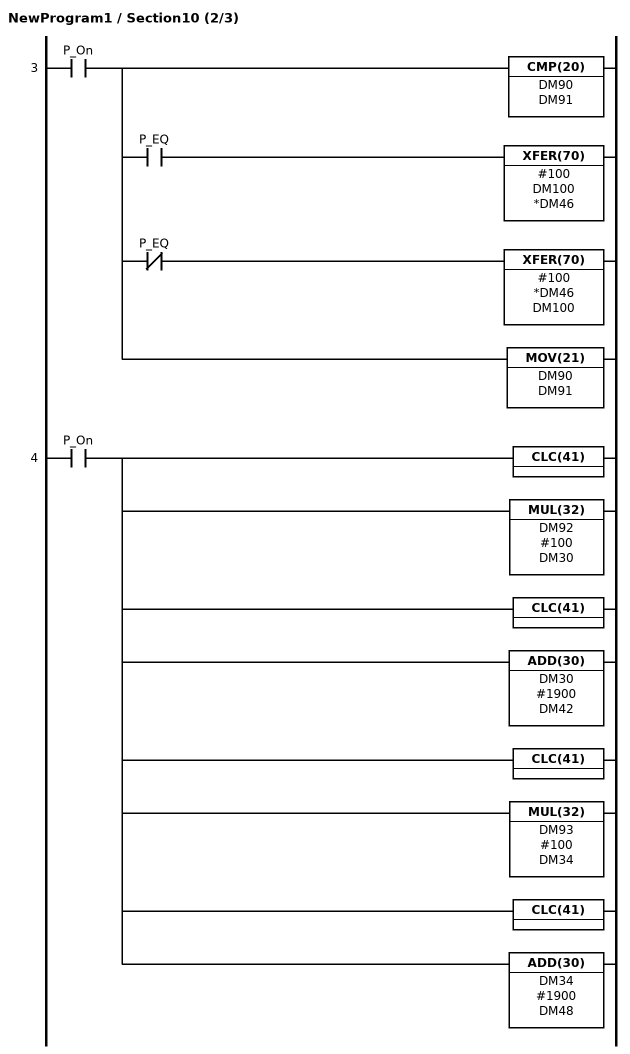
; rung 3
LD P_On
OUT TR0
CMP(20) DM90 DM91
AND P_EQ
XFER(70) #100 DM100 *DM46
LD TR0
ANDNOT P_EQ
XFER(70) #100 *DM46 DM100
LD TR0
MOV(21) DM90 DM91
; rung 4
LD P_On
CLC(41)
MUL(32) DM92 #100 DM30
CLC(41)
ADD(30) DM30 #1900 DM42
CLC(41)
MUL(32) DM93 #100 DM34
CLC(41)
ADD(30) DM34 #1900 DM48

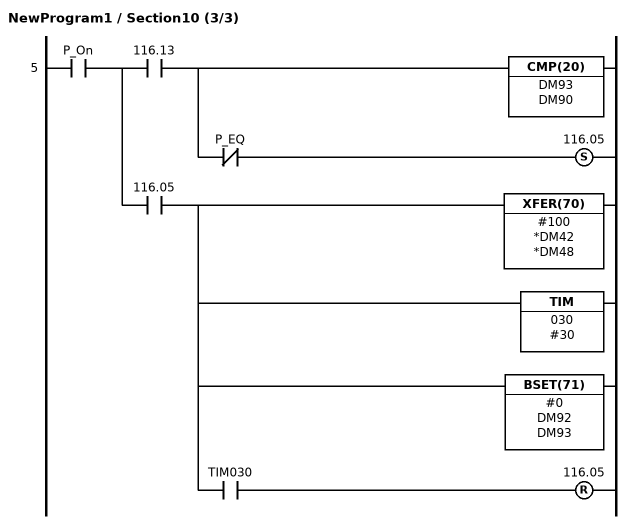
; rung 5
LD P_On
OUT TR0
AND 116.13
CMP(20) DM93 DM90
ANDNOT P_EQ
SET 116.05
LD TR0
AND 116.05
XFER(70) #100 *DM42 *DM48
TIM 030 #30
BSET(71) #0 DM92 DM93
AND TIM030
RSET 116.05

### Section Section11

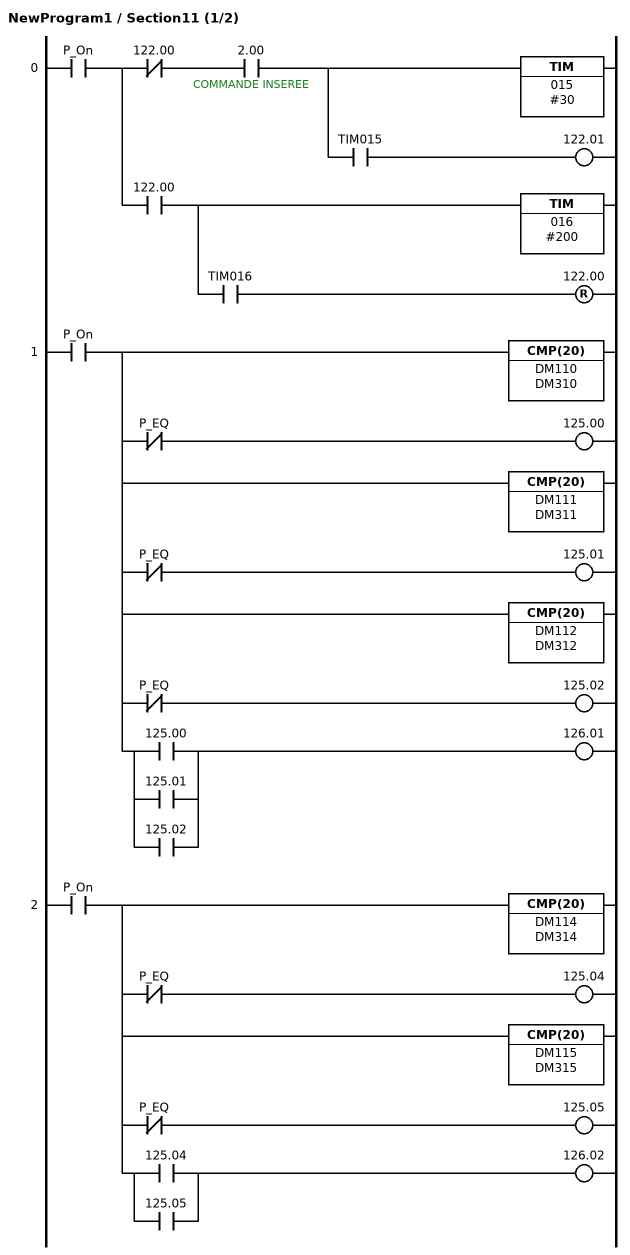
; rung 0
LD P_On
OUT TR0
ANDNOT 122.00
AND 2.00  ; COMMANDE INSEREE
TIM 015 #30
AND TIM015
OUT 122.01
LD TR0
AND 122.00
TIM 016 #200
AND TIM016
RSET 122.00
; rung 1
LD P_On
OUT TR0
CMP(20) DM110 DM310
ANDNOT P_EQ
OUT 125.00
LD TR0
CMP(20) DM111 DM311
ANDNOT P_EQ
OUT 125.01
LD TR0
CMP(20) DM112 DM312
ANDNOT P_EQ
OUT 125.02
LD TR0
LD 125.00
OR 125.01
OR 125.02
ANDLD
OUT 126.01
; rung 2
LD P_On
OUT TR0
CMP(20) DM114 DM314
ANDNOT P_EQ
OUT 125.04
LD TR0
CMP(20) DM115 DM315
ANDNOT P_EQ
OUT 125.05
LD TR0
LD 125.04
OR 125.05
ANDLD
OUT 126.02

